// TIA Portal V20 export
TYPE "LER_typeSoftCam"
// stored: Access Published
   STRUCT
      Pos0 { S7_SetPoint := 'True'} : "LER_typeSoftcamControlNodes";
      Pos1 { S7_SetPoint := 'True'} : "LER_typeSoftcamControlNodes";
      Pos2 { S7_SetPoint := 'True'} : "LER_typeSoftcamControlNodes";
      Pos3 { S7_SetPoint := 'True'} : "LER_typeSoftcamControlNodes";
      Pos4 { S7_SetPoint := 'True'} : "LER_typeSoftcamControlNodes";
      Pos5 { S7_SetPoint := 'True'} : "LER_typeSoftcamControlNodes";
      Pos6 { S7_SetPoint := 'True'} : "LER_typeSoftcamControlNodes";
      Pos7 { S7_SetPoint := 'True'} : "LER_typeSoftcamControlNodes";
      Pos8 { S7_SetPoint := 'True'} : "LER_typeSoftcamControlNodes";
      Pos9 { S7_SetPoint := 'True'} : "LER_typeSoftcamControlNodes";
      Pos10 { S7_SetPoint := 'True'} : "LER_typeSoftcamControlNodes";
      Pos11 { S7_SetPoint := 'True'} : "LER_typeSoftcamControlNodes";
      Pos12 { S7_SetPoint := 'True'} : "LER_typeSoftcamControlNodes";
      Pos13 { S7_SetPoint := 'True'} : "LER_typeSoftcamControlNodes";
      Pos14 { S7_SetPoint := 'True'} : "LER_typeSoftcamControlNodes";
      Pos15 { S7_SetPoint := 'True'} : "LER_typeSoftcamControlNodes";
   END_STRUCT;
END_TYPE
